TYPE E_Color_ARGB : CHALET_BaseComponents.E_Colors_ARGB; END_TYPE

(* stored: Version 1.1.0.1, ProductVersion 3.1.4024.12
   DUT E_Color_ARGB: Id {640c9064-9628-49d6-baf6-301282c040db} *)
